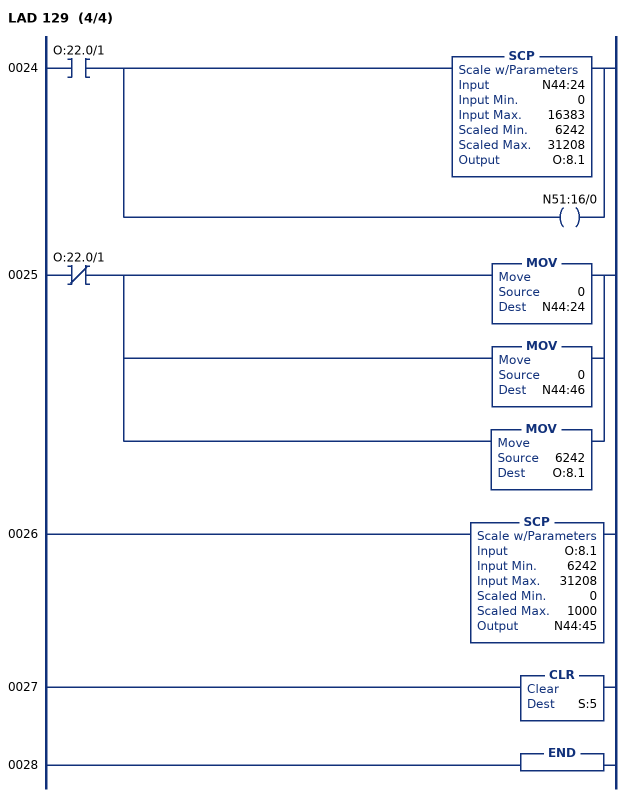
% Rung: 24 %
SOR XIC O:22.0/1 BST SCP N44:24 0 16383 6242 31208 O:8.1 NXB OTE N51:16/0 BND EOR
% Rung: 25 %
SOR XIO O:22.0/1 BST MOV 0 N44:24 NXB MOV 0 N44:46 NXB MOV 6242 O:8.1 BND EOR
% Rung: 26 %
SOR SCP O:8.1 6242 31208 0 1000 N44:45 EOR
% Rung: 27 %
SOR CLR S:5 EOR
% Rung: 28 %
SOR END EOR

LADDER 131
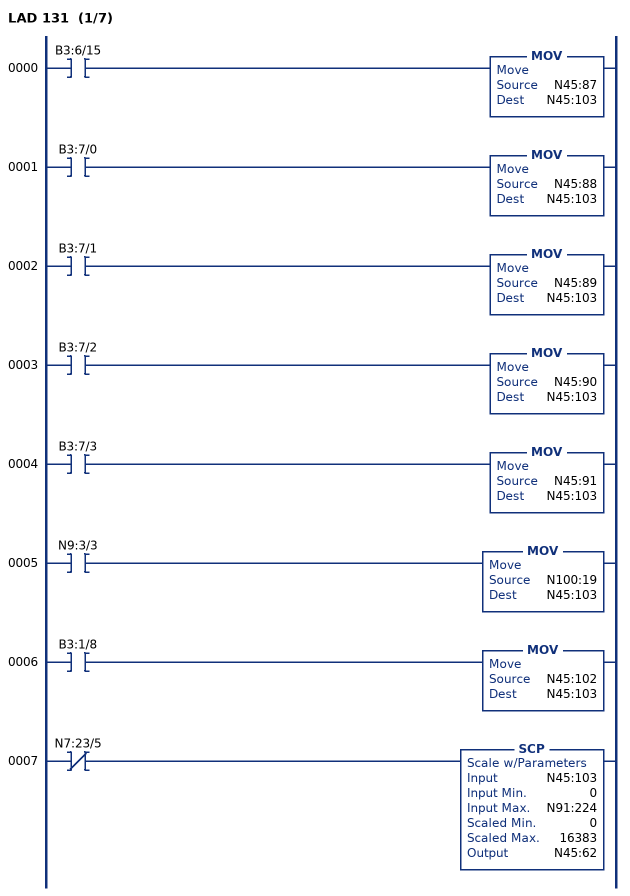
% Rung: 0 %
SOR XIC B3:6/15 MOV N45:87 N45:103 EOR
% Rung: 1 %
SOR XIC B3:7/0 MOV N45:88 N45:103 EOR
% Rung: 2 %
SOR XIC B3:7/1 MOV N45:89 N45:103 EOR
% Rung: 3 %
SOR XIC B3:7/2 MOV N45:90 N45:103 EOR
% Rung: 4 %
SOR XIC B3:7/3 MOV N45:91 N45:103 EOR
% Rung: 5 %
SOR XIC N9:3/3 MOV N100:19 N45:103 EOR
% Rung: 6 %
SOR XIC B3:1/8 MOV N45:102 N45:103 EOR
% Rung: 7 %
SOR XIO N7:23/5 SCP N45:103 0 N91:224 0 16383 N45:62 EOR

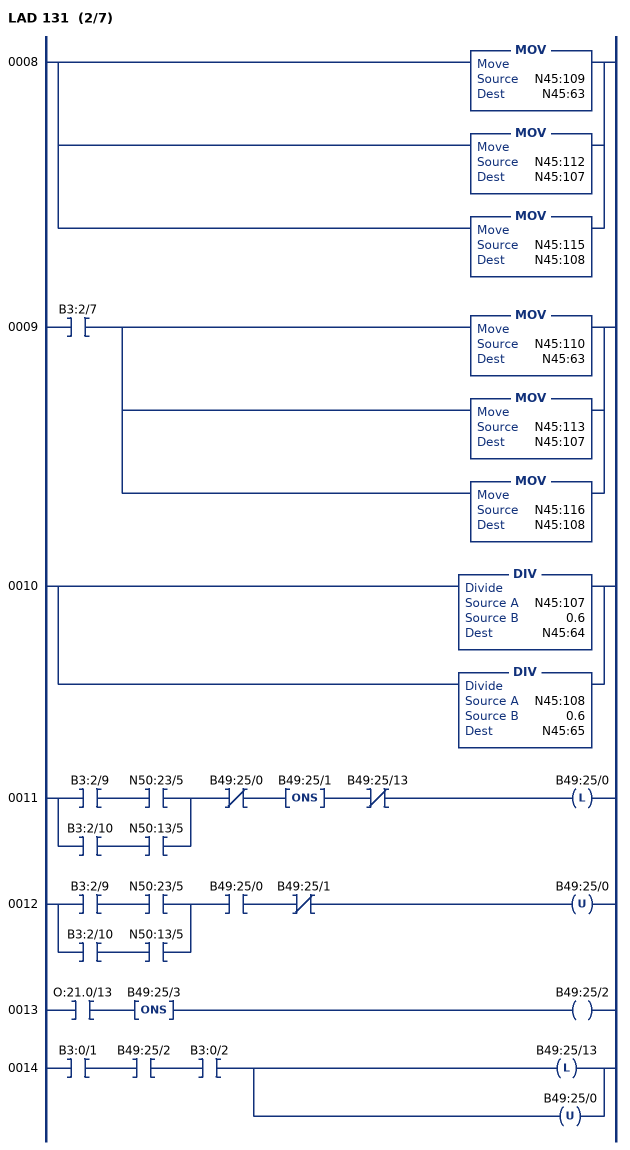
% Rung: 8 %
SOR BST MOV N45:109 N45:63 NXB MOV N45:112 N45:107 NXB MOV N45:115 N45:108 BND EOR
% Rung: 9 %
SOR XIC B3:2/7 BST MOV N45:110 N45:63 NXB MOV N45:113 N45:107 NXB MOV N45:116 N45:108 BND EOR
% Rung: 10 %
SOR BST DIV N45:107 0.6 N45:64 NXB DIV N45:108 0.6 N45:65 BND EOR
% Rung: 11 %
SOR BST XIC B3:2/9 XIC N50:23/5 NXB XIC B3:2/10 XIC N50:13/5 BND XIO B49:25/0 OSR B49:25/1 XIO B49:25/13 OTL B49:25/0 EOR
% Rung: 12 %
SOR BST XIC B3:2/9 XIC N50:23/5 NXB XIC B3:2/10 XIC N50:13/5 BND XIC B49:25/0 XIO B49:25/1 OTU B49:25/0 EOR
% Rung: 13 %
SOR XIC O:21.0/13 OSR B49:25/3 OTE B49:25/2 EOR
% Rung: 14 %
SOR XIC B3:0/1 XIC B49:25/2 XIC B3:0/2 BST OTL B49:25/13 NXB OTU B49:25/0 BND EOR

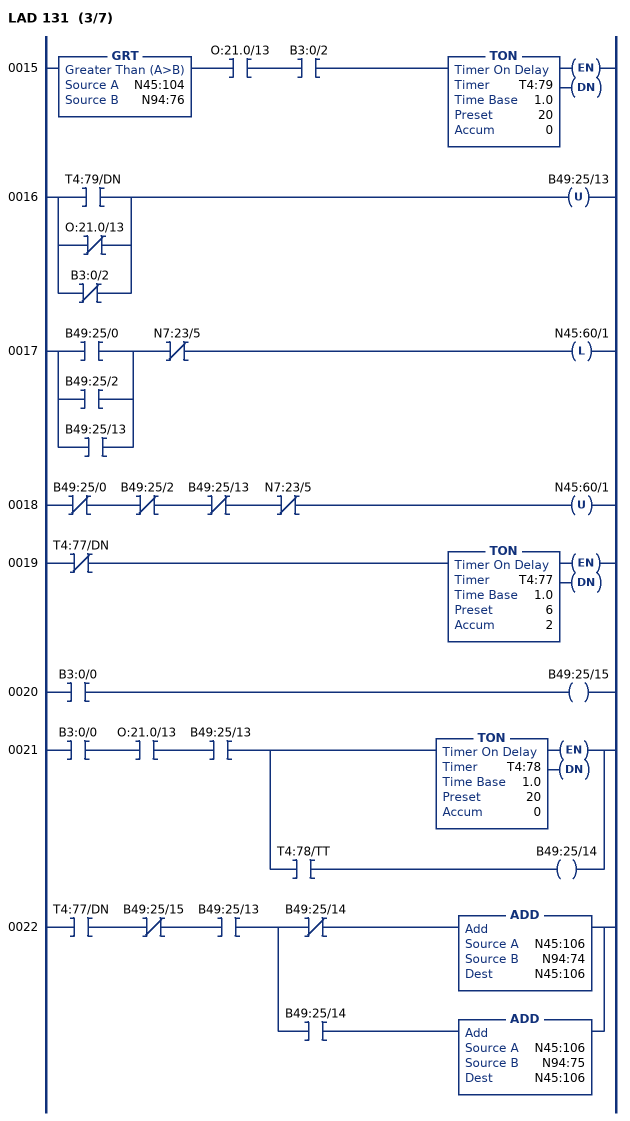
% Rung: 15 %
SOR GRT N45:104 N94:76 XIC O:21.0/13 XIC B3:0/2 TON T4:79 1.0 20 0 EOR
% Rung: 16 %
SOR BST XIC T4:79/DN NXB XIO O:21.0/13 NXB XIO B3:0/2 BND OTU B49:25/13 EOR
% Rung: 17 %
SOR BST XIC B49:25/0 NXB XIC B49:25/2 NXB XIC B49:25/13 BND XIO N7:23/5 OTL N45:60/1 EOR
% Rung: 18 %
SOR XIO B49:25/0 XIO B49:25/2 XIO B49:25/13 XIO N7:23/5 OTU N45:60/1 EOR
% Rung: 19 %
SOR XIO T4:77/DN TON T4:77 1.0 6 2 EOR
% Rung: 20 %
SOR XIC B3:0/0 OTE B49:25/15 EOR
% Rung: 21 %
SOR XIC B3:0/0 XIC O:21.0/13 XIC B49:25/13 BST TON T4:78 1.0 20 0 NXB XIC T4:78/TT OTE B49:25/14 BND EOR
% Rung: 22 %
SOR XIC T4:77/DN XIO B49:25/15 XIC B49:25/13 BST XIO B49:25/14 ADD N45:106 N94:74 N45:106 NXB XIC B49:25/14 ADD N45:106 N94:75 N45:106 BND EOR

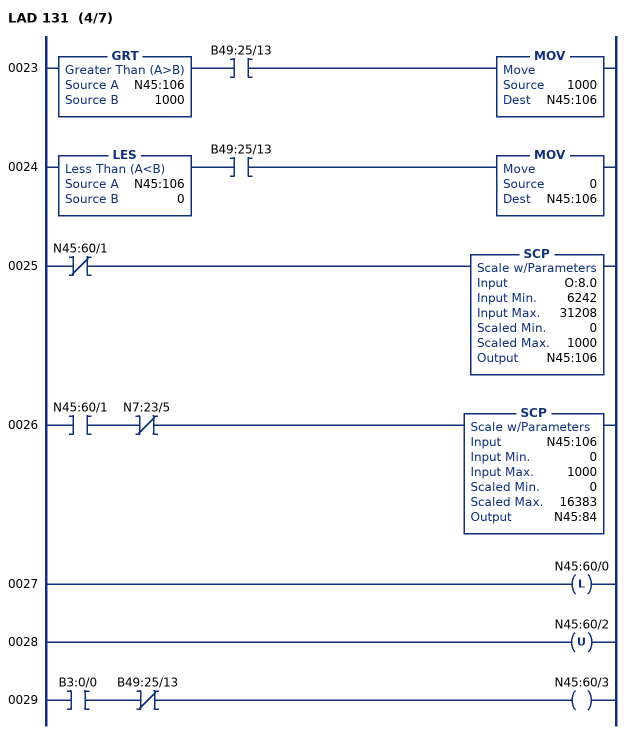
% Rung: 23 %
SOR GRT N45:106 1000 XIC B49:25/13 MOV 1000 N45:106 EOR
% Rung: 24 %
SOR LES N45:106 0 XIC B49:25/13 MOV 0 N45:106 EOR
% Rung: 25 %
SOR XIO N45:60/1 SCP O:8.0 6242 31208 0 1000 N45:106 EOR
% Rung: 26 %
SOR XIC N45:60/1 XIO N7:23/5 SCP N45:106 0 1000 0 16383 N45:84 EOR
% Rung: 27 %
SOR OTL N45:60/0 EOR
% Rung: 28 %
SOR OTU N45:60/2 EOR
% Rung: 29 %
SOR XIC B3:0/0 XIO B49:25/13 OTE N45:60/3 EOR

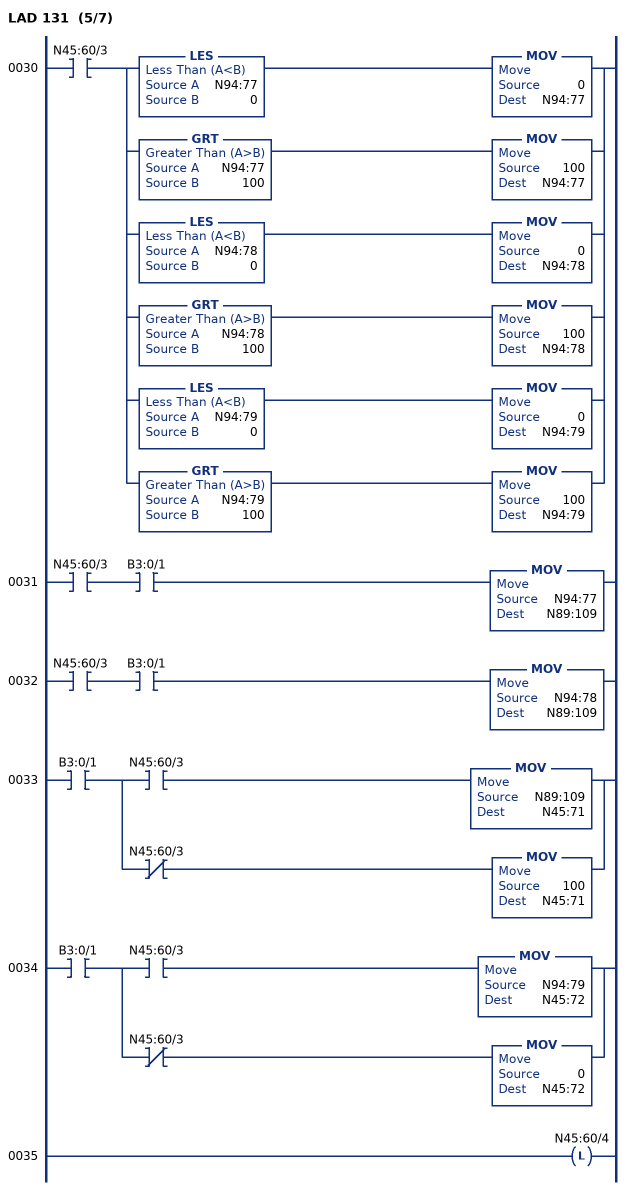
% Rung: 30 %
SOR XIC N45:60/3 BST LES N94:77 0 MOV 0 N94:77 NXB GRT N94:77 100 MOV 100 N94:77 NXB LES N94:78 0 MOV 0 N94:78 NXB GRT N94:78 100 MOV 100 N94:78 NXB LES N94:79 0 MOV 0 N94:79 NXB GRT N94:79 100 MOV 100 N94:79 BND EOR
% Rung: 31 %
SOR XIC N45:60/3 XIC B3:0/1 MOV N94:77 N89:109 EOR
% Rung: 32 %
SOR XIC N45:60/3 XIC B3:0/1 MOV N94:78 N89:109 EOR
% Rung: 33 %
SOR XIC B3:0/1 BST XIC N45:60/3 MOV N89:109 N45:71 NXB XIO N45:60/3 MOV 100 N45:71 BND EOR
% Rung: 34 %
SOR XIC B3:0/1 BST XIC N45:60/3 MOV N94:79 N45:72 NXB XIO N45:60/3 MOV 0 N45:72 BND EOR
% Rung: 35 %
SOR OTL N45:60/4 EOR

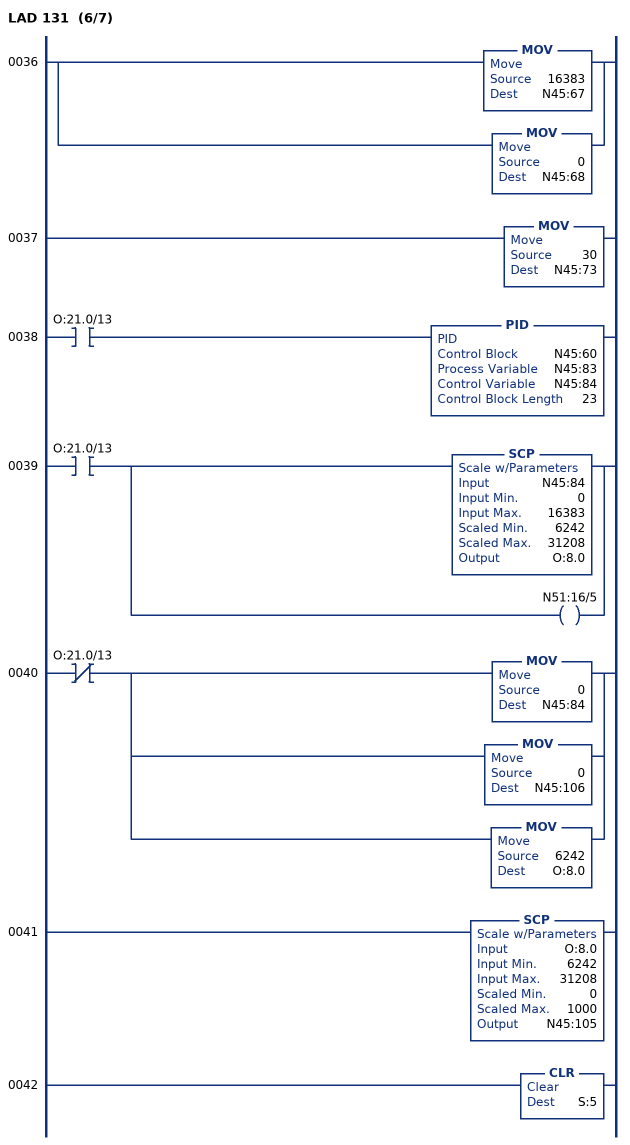
% Rung: 36 %
SOR BST MOV 16383 N45:67 NXB MOV 0 N45:68 BND EOR
% Rung: 37 %
SOR MOV 30 N45:73 EOR
% Rung: 38 %
SOR XIC O:21.0/13 PID N45:60 N45:83 N45:84 23 EOR
% Rung: 39 %
SOR XIC O:21.0/13 BST SCP N45:84 0 16383 6242 31208 O:8.0 NXB OTE N51:16/5 BND EOR
% Rung: 40 %
SOR XIO O:21.0/13 BST MOV 0 N45:84 NXB MOV 0 N45:106 NXB MOV 6242 O:8.0 BND EOR
% Rung: 41 %
SOR SCP O:8.0 6242 31208 0 1000 N45:105 EOR
% Rung: 42 %
SOR CLR S:5 EOR

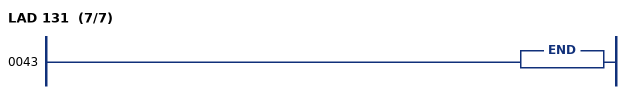
% Rung: 43 %
SOR END EOR

LADDER 132
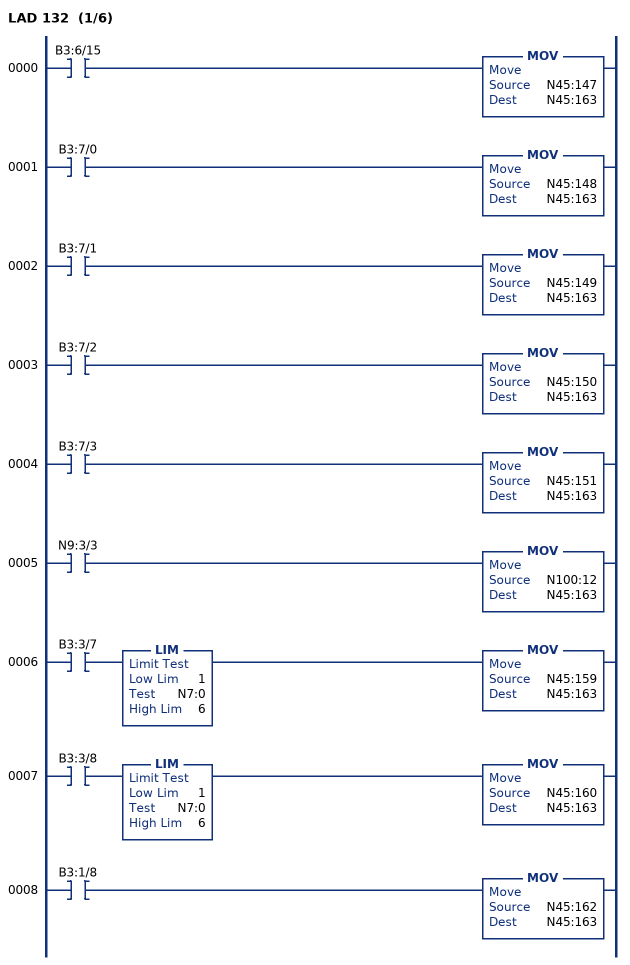
% Rung: 0 %
SOR XIC B3:6/15 MOV N45:147 N45:163 EOR
% Rung: 1 %
SOR XIC B3:7/0 MOV N45:148 N45:163 EOR
% Rung: 2 %
SOR XIC B3:7/1 MOV N45:149 N45:163 EOR
% Rung: 3 %
SOR XIC B3:7/2 MOV N45:150 N45:163 EOR
% Rung: 4 %
SOR XIC B3:7/3 MOV N45:151 N45:163 EOR
% Rung: 5 %
SOR XIC N9:3/3 MOV N100:12 N45:163 EOR
% Rung: 6 %
SOR XIC B3:3/7 LIM 1 N7:0 6 MOV N45:159 N45:163 EOR
% Rung: 7 %
SOR XIC B3:3/8 LIM 1 N7:0 6 MOV N45:160 N45:163 EOR
% Rung: 8 %
SOR XIC B3:1/8 MOV N45:162 N45:163 EOR

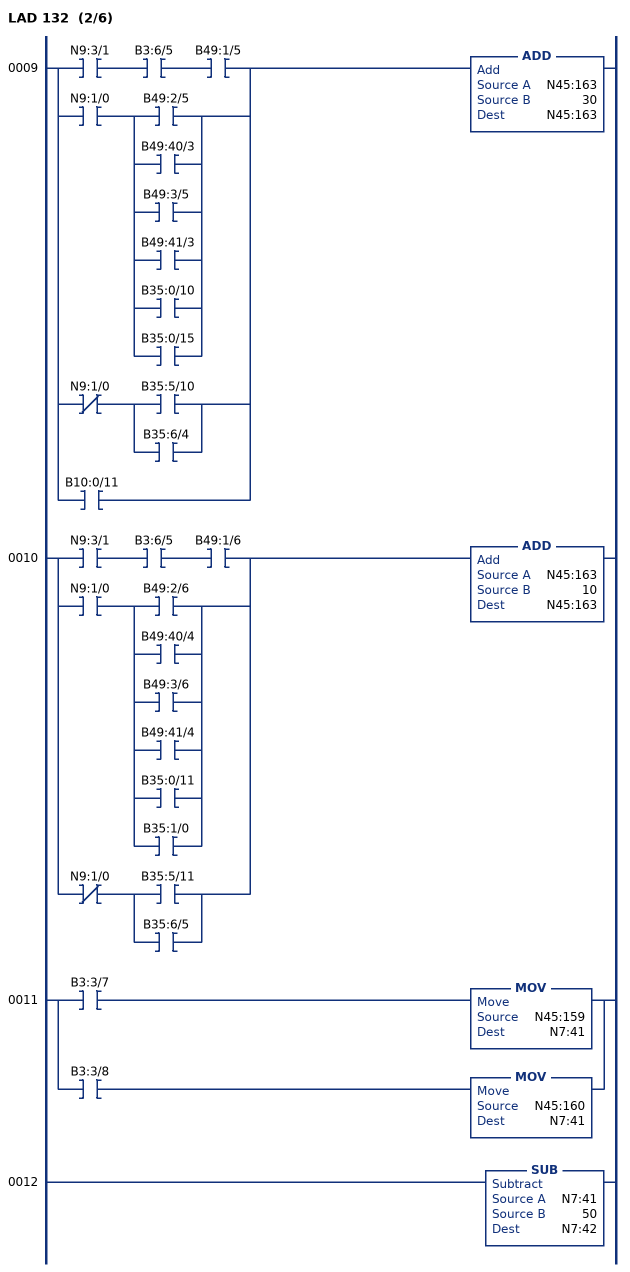
% Rung: 9 %
SOR BST XIC N9:3/1 XIC B3:6/5 XIC B49:1/5 NXB XIC N9:1/0 BST XIC B49:2/5 NXB XIC B49:40/3 NXB XIC B49:3/5 NXB XIC B49:41/3 NXB XIC B35:0/10 NXB XIC B35:0/15 BND NXB XIO N9:1/0 BST XIC B35:5/10 NXB XIC B35:6/4 BND NXB XIC B10:0/11 BND ADD N45:163 30 N45:163 EOR
% Rung: 10 %
SOR BST XIC N9:3/1 XIC B3:6/5 XIC B49:1/6 NXB XIC N9:1/0 BST XIC B49:2/6 NXB XIC B49:40/4 NXB XIC B49:3/6 NXB XIC B49:41/4 NXB XIC B35:0/11 NXB XIC B35:1/0 BND NXB XIO N9:1/0 BST XIC B35:5/11 NXB XIC B35:6/5 BND BND ADD N45:163 10 N45:163 EOR
% Rung: 11 %
SOR BST XIC B3:3/7 MOV N45:159 N7:41 NXB XIC B3:3/8 MOV N45:160 N7:41 BND EOR
% Rung: 12 %
SOR SUB N7:41 50 N7:42 EOR

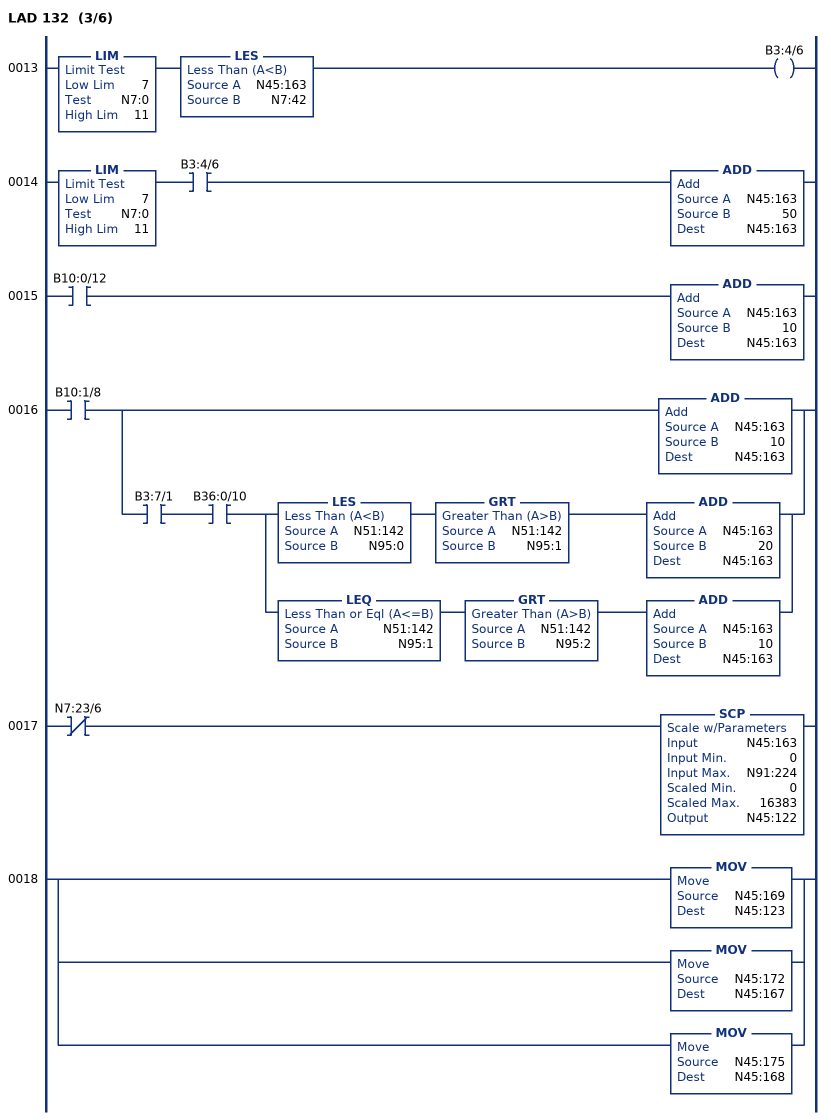
% Rung: 13 %
SOR LIM 7 N7:0 11 LES N45:163 N7:42 OTE B3:4/6 EOR
% Rung: 14 %
SOR LIM 7 N7:0 11 XIC B3:4/6 ADD N45:163 50 N45:163 EOR
% Rung: 15 %
SOR XIC B10:0/12 ADD N45:163 10 N45:163 EOR
% Rung: 16 %
SOR XIC B10:1/8 BST ADD N45:163 10 N45:163 NXB XIC B3:7/1 XIC B36:0/10 BST LES N51:142 N95:0 GRT N51:142 N95:1 ADD N45:163 20 N45:163 NXB LEQ N51:142 N95:1 GRT N51:142 N95:2 ADD N45:163 10 N45:163 BND BND EOR
% Rung: 17 %
SOR XIO N7:23/6 SCP N45:163 0 N91:224 0 16383 N45:122 EOR
% Rung: 18 %
SOR BST MOV N45:169 N45:123 NXB MOV N45:172 N45:167 NXB MOV N45:175 N45:168 BND EOR

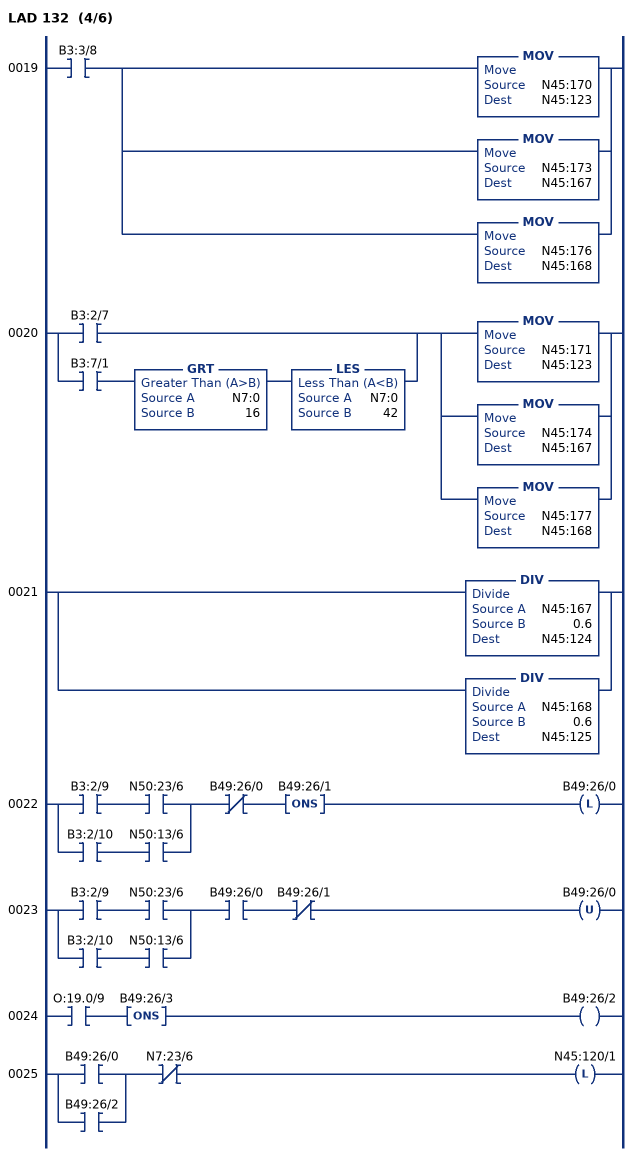
% Rung: 19 %
SOR XIC B3:3/8 BST MOV N45:170 N45:123 NXB MOV N45:173 N45:167 NXB MOV N45:176 N45:168 BND EOR
% Rung: 20 %
SOR BST XIC B3:2/7 NXB XIC B3:7/1 GRT N7:0 16 LES N7:0 42 BND BST MOV N45:171 N45:123 NXB MOV N45:174 N45:167 NXB MOV N45:177 N45:168 BND EOR
% Rung: 21 %
SOR BST DIV N45:167 0.6 N45:124 NXB DIV N45:168 0.6 N45:125 BND EOR
% Rung: 22 %
SOR BST XIC B3:2/9 XIC N50:23/6 NXB XIC B3:2/10 XIC N50:13/6 BND XIO B49:26/0 OSR B49:26/1 OTL B49:26/0 EOR
% Rung: 23 %
SOR BST XIC B3:2/9 XIC N50:23/6 NXB XIC B3:2/10 XIC N50:13/6 BND XIC B49:26/0 XIO B49:26/1 OTU B49:26/0 EOR
% Rung: 24 %
SOR XIC O:19.0/9 OSR B49:26/3 OTE B49:26/2 EOR
% Rung: 25 %
SOR BST XIC B49:26/0 NXB XIC B49:26/2 BND XIO N7:23/6 OTL N45:120/1 EOR

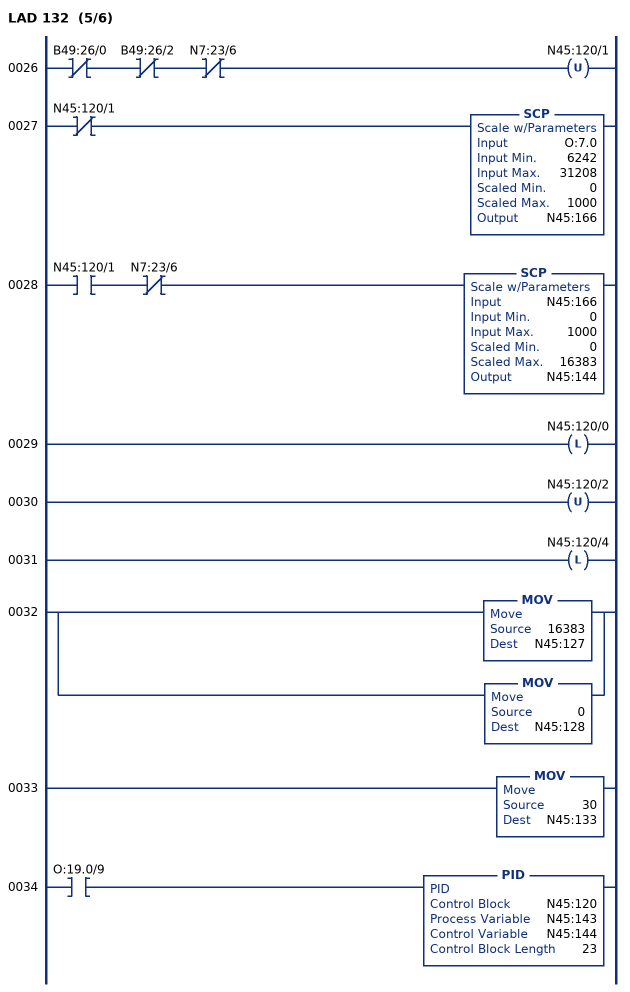
% Rung: 26 %
SOR XIO B49:26/0 XIO B49:26/2 XIO N7:23/6 OTU N45:120/1 EOR
% Rung: 27 %
SOR XIO N45:120/1 SCP O:7.0 6242 31208 0 1000 N45:166 EOR
% Rung: 28 %
SOR XIC N45:120/1 XIO N7:23/6 SCP N45:166 0 1000 0 16383 N45:144 EOR
% Rung: 29 %
SOR OTL N45:120/0 EOR
% Rung: 30 %
SOR OTU N45:120/2 EOR
% Rung: 31 %
SOR OTL N45:120/4 EOR
% Rung: 32 %
SOR BST MOV 16383 N45:127 NXB MOV 0 N45:128 BND EOR
% Rung: 33 %
SOR MOV 30 N45:133 EOR
% Rung: 34 %
SOR XIC O:19.0/9 PID N45:120 N45:143 N45:144 23 EOR

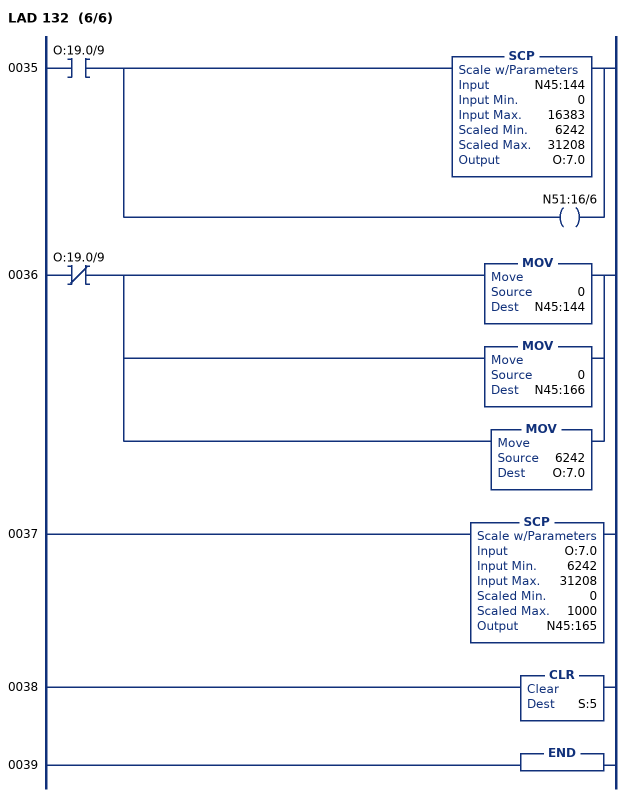
% Rung: 35 %
SOR XIC O:19.0/9 BST SCP N45:144 0 16383 6242 31208 O:7.0 NXB OTE N51:16/6 BND EOR
% Rung: 36 %
SOR XIO O:19.0/9 BST MOV 0 N45:144 NXB MOV 0 N45:166 NXB MOV 6242 O:7.0 BND EOR
% Rung: 37 %
SOR SCP O:7.0 6242 31208 0 1000 N45:165 EOR
% Rung: 38 %
SOR CLR S:5 EOR
% Rung: 39 %
SOR END EOR

LADDER 133
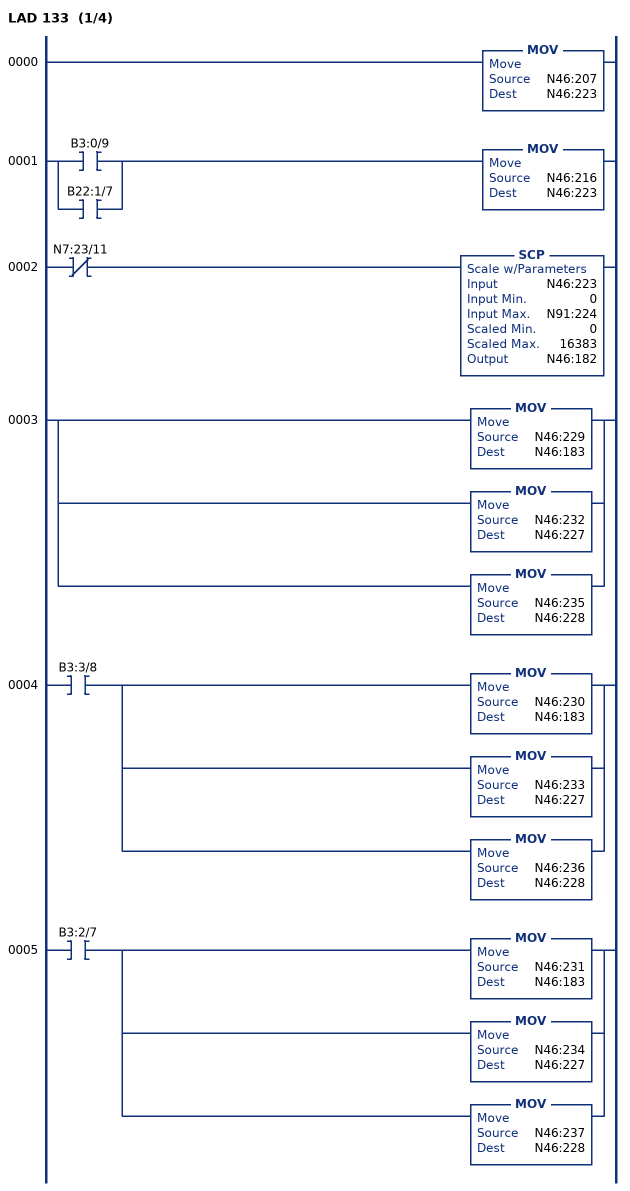
% Rung: 0 %
SOR MOV N46:207 N46:223 EOR
% Rung: 1 %
SOR BST XIC B3:0/9 NXB XIC B22:1/7 BND MOV N46:216 N46:223 EOR
% Rung: 2 %
SOR XIO N7:23/11 SCP N46:223 0 N91:224 0 16383 N46:182 EOR
% Rung: 3 %
SOR BST MOV N46:229 N46:183 NXB MOV N46:232 N46:227 NXB MOV N46:235 N46:228 BND EOR
% Rung: 4 %
SOR XIC B3:3/8 BST MOV N46:230 N46:183 NXB MOV N46:233 N46:227 NXB MOV N46:236 N46:228 BND EOR
% Rung: 5 %
SOR XIC B3:2/7 BST MOV N46:231 N46:183 NXB MOV N46:234 N46:227 NXB MOV N46:237 N46:228 BND EOR

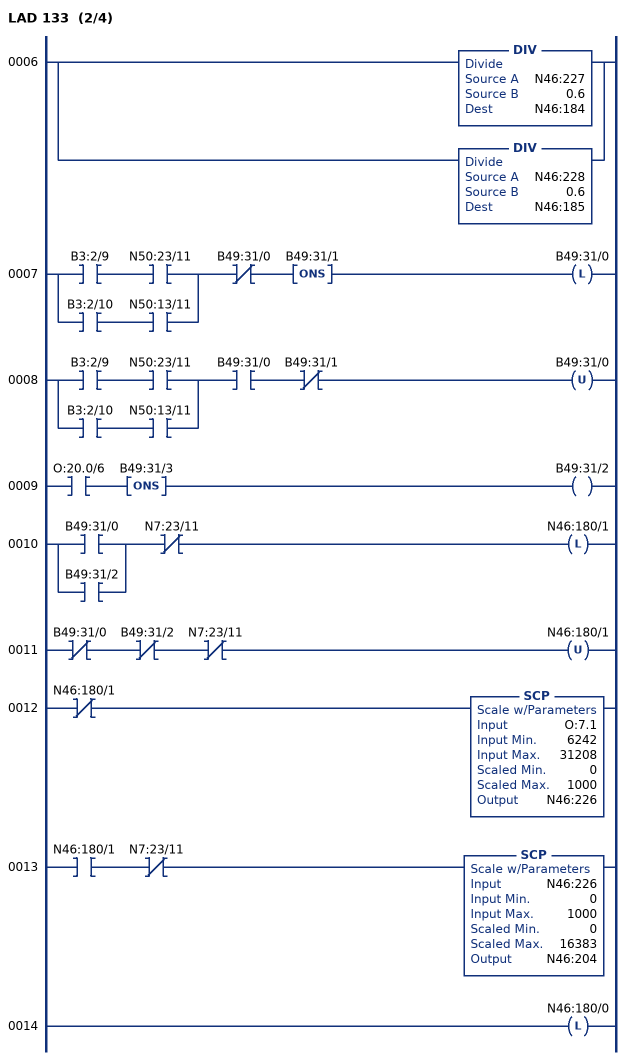
% Rung: 6 %
SOR BST DIV N46:227 0.6 N46:184 NXB DIV N46:228 0.6 N46:185 BND EOR
% Rung: 7 %
SOR BST XIC B3:2/9 XIC N50:23/11 NXB XIC B3:2/10 XIC N50:13/11 BND XIO B49:31/0 OSR B49:31/1 OTL B49:31/0 EOR
% Rung: 8 %
SOR BST XIC B3:2/9 XIC N50:23/11 NXB XIC B3:2/10 XIC N50:13/11 BND XIC B49:31/0 XIO B49:31/1 OTU B49:31/0 EOR
% Rung: 9 %
SOR XIC O:20.0/6 OSR B49:31/3 OTE B49:31/2 EOR
% Rung: 10 %
SOR BST XIC B49:31/0 NXB XIC B49:31/2 BND XIO N7:23/11 OTL N46:180/1 EOR
% Rung: 11 %
SOR XIO B49:31/0 XIO B49:31/2 XIO N7:23/11 OTU N46:180/1 EOR
% Rung: 12 %
SOR XIO N46:180/1 SCP O:7.1 6242 31208 0 1000 N46:226 EOR
% Rung: 13 %
SOR XIC N46:180/1 XIO N7:23/11 SCP N46:226 0 1000 0 16383 N46:204 EOR
% Rung: 14 %
SOR OTL N46:180/0 EOR

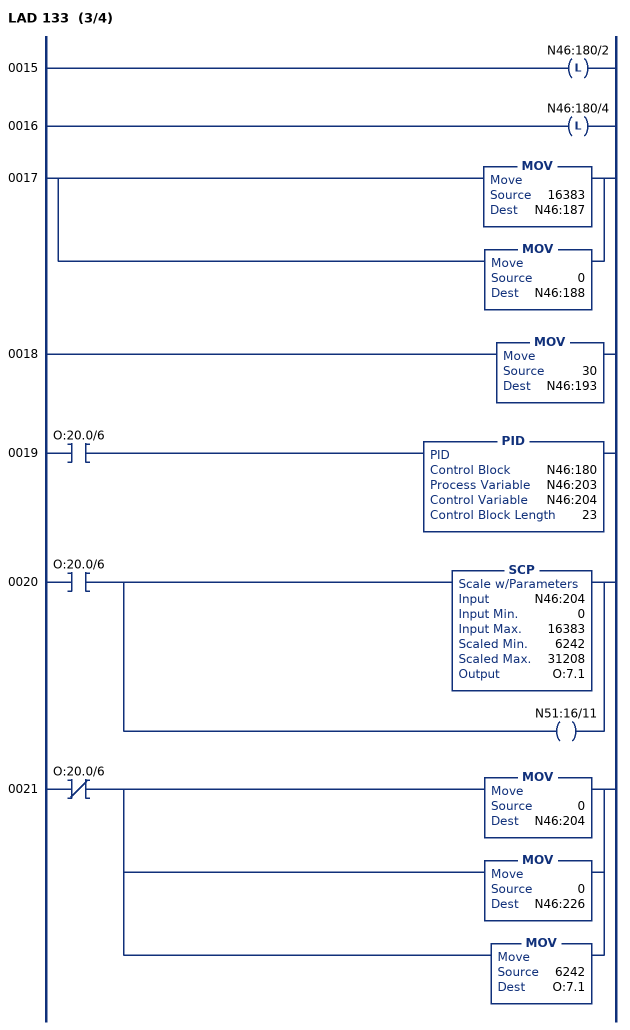
% Rung: 15 %
SOR OTL N46:180/2 EOR
% Rung: 16 %
SOR OTL N46:180/4 EOR
% Rung: 17 %
SOR BST MOV 16383 N46:187 NXB MOV 0 N46:188 BND EOR
% Rung: 18 %
SOR MOV 30 N46:193 EOR
% Rung: 19 %
SOR XIC O:20.0/6 PID N46:180 N46:203 N46:204 23 EOR
% Rung: 20 %
SOR XIC O:20.0/6 BST SCP N46:204 0 16383 6242 31208 O:7.1 NXB OTE N51:16/11 BND EOR
% Rung: 21 %
SOR XIO O:20.0/6 BST MOV 0 N46:204 NXB MOV 0 N46:226 NXB MOV 6242 O:7.1 BND EOR

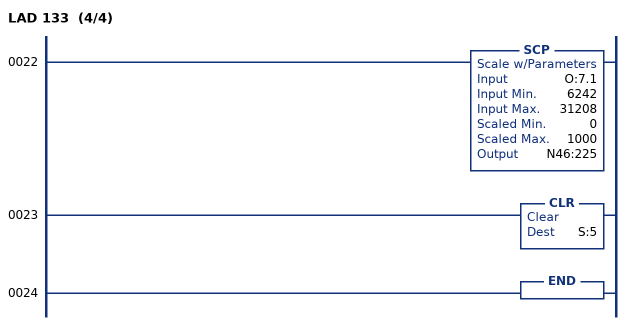
% Rung: 22 %
SOR SCP O:7.1 6242 31208 0 1000 N46:225 EOR
% Rung: 23 %
SOR CLR S:5 EOR
% Rung: 24 %
SOR END EOR

LADDER 134
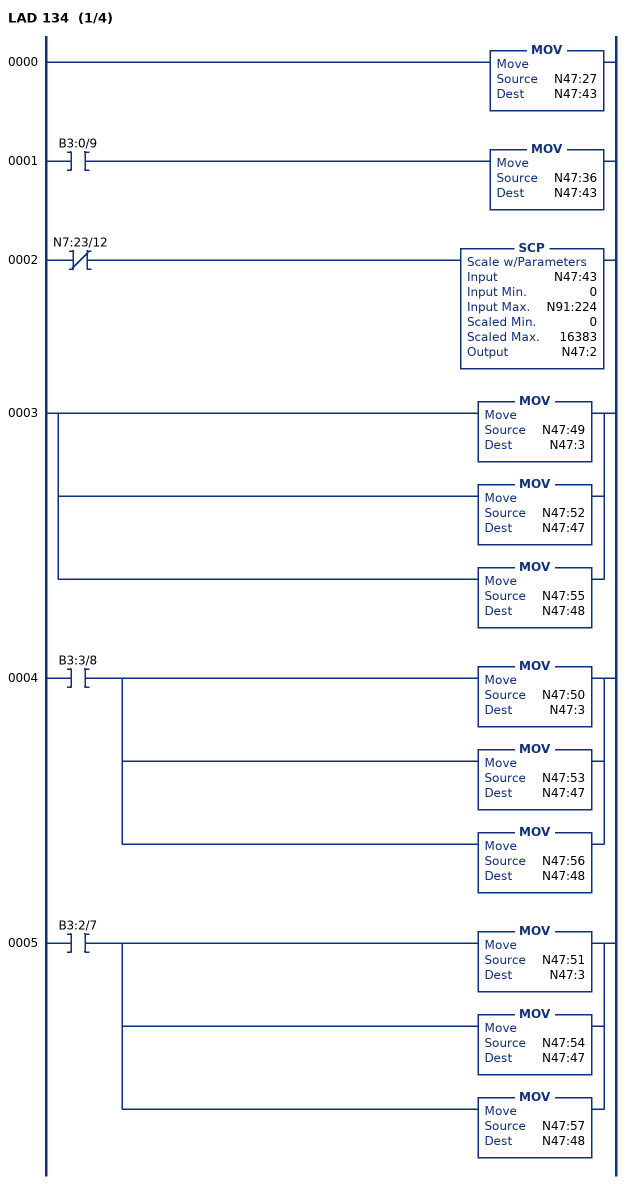
% Rung: 0 %
SOR MOV N47:27 N47:43 EOR
% Rung: 1 %
SOR XIC B3:0/9 MOV N47:36 N47:43 EOR
% Rung: 2 %
SOR XIO N7:23/12 SCP N47:43 0 N91:224 0 16383 N47:2 EOR
% Rung: 3 %
SOR BST MOV N47:49 N47:3 NXB MOV N47:52 N47:47 NXB MOV N47:55 N47:48 BND EOR
% Rung: 4 %
SOR XIC B3:3/8 BST MOV N47:50 N47:3 NXB MOV N47:53 N47:47 NXB MOV N47:56 N47:48 BND EOR
% Rung: 5 %
SOR XIC B3:2/7 BST MOV N47:51 N47:3 NXB MOV N47:54 N47:47 NXB MOV N47:57 N47:48 BND EOR

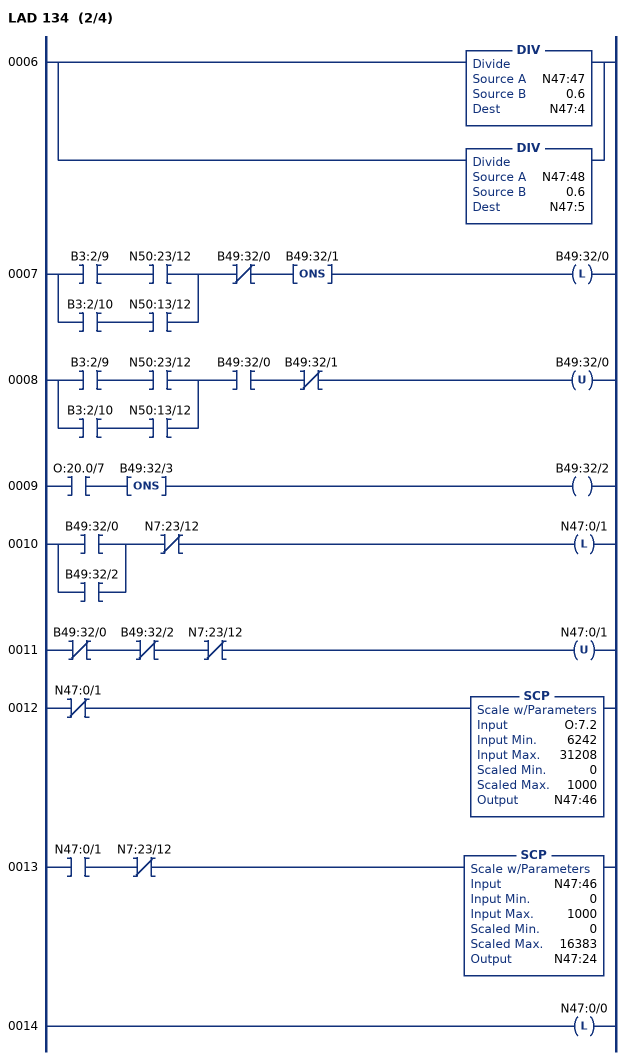
% Rung: 6 %
SOR BST DIV N47:47 0.6 N47:4 NXB DIV N47:48 0.6 N47:5 BND EOR
% Rung: 7 %
SOR BST XIC B3:2/9 XIC N50:23/12 NXB XIC B3:2/10 XIC N50:13/12 BND XIO B49:32/0 OSR B49:32/1 OTL B49:32/0 EOR
% Rung: 8 %
SOR BST XIC B3:2/9 XIC N50:23/12 NXB XIC B3:2/10 XIC N50:13/12 BND XIC B49:32/0 XIO B49:32/1 OTU B49:32/0 EOR
% Rung: 9 %
SOR XIC O:20.0/7 OSR B49:32/3 OTE B49:32/2 EOR
% Rung: 10 %
SOR BST XIC B49:32/0 NXB XIC B49:32/2 BND XIO N7:23/12 OTL N47:0/1 EOR
% Rung: 11 %
SOR XIO B49:32/0 XIO B49:32/2 XIO N7:23/12 OTU N47:0/1 EOR
% Rung: 12 %
SOR XIO N47:0/1 SCP O:7.2 6242 31208 0 1000 N47:46 EOR
% Rung: 13 %
SOR XIC N47:0/1 XIO N7:23/12 SCP N47:46 0 1000 0 16383 N47:24 EOR
% Rung: 14 %
SOR OTL N47:0/0 EOR

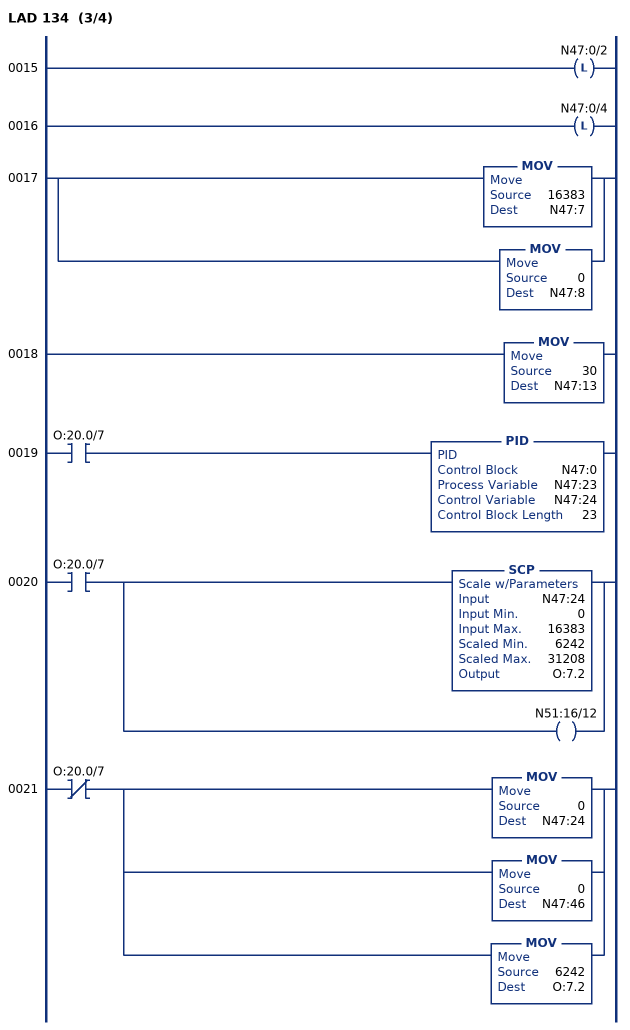
% Rung: 15 %
SOR OTL N47:0/2 EOR
% Rung: 16 %
SOR OTL N47:0/4 EOR
% Rung: 17 %
SOR BST MOV 16383 N47:7 NXB MOV 0 N47:8 BND EOR
% Rung: 18 %
SOR MOV 30 N47:13 EOR
% Rung: 19 %
SOR XIC O:20.0/7 PID N47:0 N47:23 N47:24 23 EOR
% Rung: 20 %
SOR XIC O:20.0/7 BST SCP N47:24 0 16383 6242 31208 O:7.2 NXB OTE N51:16/12 BND EOR
% Rung: 21 %
SOR XIO O:20.0/7 BST MOV 0 N47:24 NXB MOV 0 N47:46 NXB MOV 6242 O:7.2 BND EOR

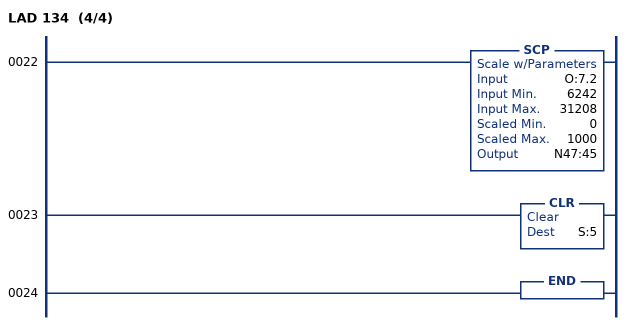
% Rung: 22 %
SOR SCP O:7.2 6242 31208 0 1000 N47:45 EOR
% Rung: 23 %
SOR CLR S:5 EOR
% Rung: 24 %
SOR END EOR

DATA TABLE (non-zero values as saved)
DATA B3
% B3:0 % 0X0002 0X0841 0X0300 0X0084 0X3F80 0X8000 0X8540 0X0000 0X0000 0X0000
% B3:10 % 0X0001 0X0000 0X0000 0X0000 0X0000 0X0000 0X0000 0X0000 0X0000 0X0401
% B3:20 % 0X0000 0X0000 0X0000 0X0000 0X0000 0X00A6 0X0000 0X0000 0X0000 0X0000
% B3:40 % 0X0000 0X0001 0X0000 0X0000 0X0000 0X0000 0X0000 0X0000 0X0000 0X0000
% B3:60 % 0X0000 0X0004 0X0020 0X0000 0X0800 0X0002 0X0000 0X00FE 0X0000 0X0000
% B3:70 % 0X0040 0X0000 0X8000 0X0001 0X0000 0X0000 0X0000 0X0000 0X0000 0X0000
% B3:120 % 0X0000 0X0000 0X0000 0X0000 0X0000 0X0000 0X8000 0X0000 0X0000 0X0000
DATA T4
% .PRE .ACC %
% T4:1 % 15 13
% T4:3 % 50 38
% T4:4 % 50 0
% T4:5 % 15 0
% T4:6 % 60 0
% T4:7 % 120 120
% T4:8 % 3600 0
% T4:9 % 30000 0
% T4:10 % 30 0
% T4:11 % 500 0
% T4:12 % 10 0
% T4:13 % 10 0
% T4:14 % 200 0
% T4:15 % 60 0
% T4:16 % 50 0
% T4:17 % 100 0
% T4:18 % 30 0
% T4:20 % 1 0
% T4:21 % 60 20
% T4:22 % 3 3
% T4:25 % 25 0
% T4:26 % 30 0
% T4:30 % 25 25
% T4:31 % 10 0
% T4:32 % 5 5
% T4:33 % 300 0
% T4:34 % 30 0
% T4:35 % 1 0
% T4:36 % 30 0
% T4:37 % 10 0
% T4:38 % 1 0
% T4:40 % 20 0
% T4:41 % 20 0
% T4:42 % 200 0
% T4:43 % 100 100
% T4:44 % 50 0
% T4:49 % 30 0
% T4:50 % 1 0
% T4:51 % 20 0
% T4:52 % 6 5
% T4:53 % 20 0
% T4:54 % 20 20
% T4:55 % 1 0
% T4:56 % 20 0
% T4:60 % 150 0
% T4:61 % 20 0
% T4:65 % 1 0
% T4:66 % 20 0
% T4:72 % 6 6
% T4:73 % 20 0
% T4:74 % 20 0
% T4:75 % 20 0
% T4:77 % 6 2
% T4:78 % 20 0
% T4:79 % 20 0
% T4:80 % 1 0
% T4:81 % 20 0
% T4:85 % 1 0
% T4:86 % 20 0
% T4:90 % 1 0
% T4:91 % 20 0
% T4:92 % 1 0
% T4:93 % 20 0
% T4:100 % 1 0
% T4:101 % 20 0
% T4:111 % 120 0
% T4:112 % 6 6
% T4:113 % 20 0
% T4:114 % 20 0
% T4:115 % 222 0
% T4:116 % 6 6
% T4:117 % 20 0
% T4:119 % 60 0
% T4:120 % 6 6
% T4:121 % 20 0
DATA C5
% .PRE .ACC %
% C5:0 % 4 0
% C5:1 % 2 0
% C5:4 % 2 0
% C5:5 % 3 0
DATA R6
% .LEN .POS %
% R6:0 % 3 0
% R6:1 % 4 0
% R6:2 % 4 0
% R6:3 % 3 0
% R6:4 % 14 0
% R6:5 % 14 0
% R6:6 % 14 0
% R6:7 % 14 0
% R6:8 % 14 0
% R6:9 % 14 0
% R6:10 % 14 0
% R6:11 % 14 0
DATA N7
% N7:0 % 0 514 200 0 0 11 101 10 0 0
% N7:10 % 0 514 200 0 0 0 0 0 0 0
% N7:30 % 1390 0 0 0 0 0 0 0 0 0
% N7:40 % -1 1380 1330 0 0 0 0 0 0 0
% N7:50 % 0 14 0
DATA F8
% F8:0 % 237.777 0 0 0 0
% F8:5 % 0 0.01 0 0 0
% F8:10 % 1 770 1 900 1
% F8:15 % 950 0 0 1 1000
% F8:20 % 1 820 1 0 0.7076923
% F8:25 % 0 1.25 630 0.7076923 0
% F8:30 % 1 1000 1 0 1
% F8:35 % 0 1 0 2 150
% F8:40 % 17.87234 0 0 0 0
DATA N9
% N9:0 % 18434 2683 699 4243 0 0 0 0 0 2
% N9:10 % 2957 0 0 0
DATA B10
% B10:0 % 0X0001 0X0000 0X0000 0X0000 0X0000 0X0000 0X0000 0X0000 0X0000 0X0000
DATA B11
% B11:0 % 0X0001 0X0000 0X0000 0X0000 0X0000 0X0000 0X0000 0X0000 0X0000 0X0000
% B11:30 % 0X0000 0X0000 0X0004
DATA B12
% B12:0 % 0X0001 0X0000 0X0000 0X0000 0X0000 0X0000 0X0000 0X0000 0X0000 0X0000
% B12:10 % 0X0000 0X0000 0X0100 0X0000
DATA B18
% B18:0 % 0X0000 0X0010 0X0000 0X0000
DATA T21
% .PRE .ACC %
% T21:1 % 5 0
% T21:2 % 5 0
% T21:3 % 5 0
% T21:4 % 5 0
% T21:5 % 5 0
% T21:6 % 25 0
% T21:7 % 5 0
% T21:8 % 5 0
% T21:9 % 5 0
% T21:10 % 5 0
% T21:11 % 5 0
% T21:12 % 5 0
% T21:13 % 5 0
% T21:14 % 5 0
% T21:15 % 15 0
% T21:16 % 5 0
% T21:17 % 1000 0
% T21:18 % 600 0
% T21:19 % 10 0
% T21:20 % 10 0
% T21:21 % 300 0
% T21:22 % 1200 0
% T21:23 % 300 0
% T21:24 % 5 0
% T21:25 % 1 0
% T21:27 % 15 0
% T21:28 % 15 0
% T21:29 % 15 0
% T21:30 % 15 0
% T21:31 % 1200 0
% T21:32 % 600 0
% T21:33 % 300 0
% T21:34 % 15 0
% T21:35 % 1 0
% T21:36 % 10 0
% T21:37 % 600 0
% T21:38 % 180 0
% T21:40 % 600 0
% T21:41 % 20 0
% T21:42 % 10 0
% T21:43 % 120 0
% T21:44 % 120 0
% T21:45 % 60 0
% T21:46 % 1 1
% T21:47 % 5 0
% T21:48 % 1 1
% T21:49 % 1 1
% T21:50 % 120 0
% T21:51 % 10 0
% T21:52 % 10 0
% T21:53 % 5 0
% T21:54 % 50 54
% T21:55 % 50 50
% T21:56 % 50 50
% T21:57 % 50 50
% T21:58 % 50 50
% T21:59 % 50 50
% T21:61 % 10 0
% T21:62 % 2 0
% T21:63 % 4 0
% T21:70 % 2 0
% T21:71 % 5 0
% T21:72 % 5 0
% T21:73 % 5 0
% T21:74 % 600 0
% T21:75 % 20 0
% T21:76 % 5 0
% T21:77 % 5 0
% T21:78 % 5 0
% T21:79 % 5 0
% T21:80 % 5 0
% T21:81 % 15 0
% T21:84 % 5 0
DATA B24
% B24:0 % 0X0000 0X0000 0X0000 0X0004 0X0000 0X0000 0X0010 0X0000
DATA N25
% N25:0 % 244 1350 1350 1000 1350 1330 1330 1300 1100 0
% N25:20 % 294 1250 1250 1100 500 450 350 350 950 400
% N25:40 % 0 950 950 950 950 950 950 0 0 0
% N25:60 % 0 950 950 950 950 950 950 0 0 0
% N25:80 % 0 950 950 950 950 950 950 0 0 0
% N25:100 % 0 100 0 0 0 0 0 0 0 0
% N25:110 % 1 50 50 400 300 400 0 0 0 0
% N25:120 % 0 0 0 15400 14600 900 700 0 0 0
% N25:130 % 0 0 0 20426 20326 0 0 0 0 0
% N25:140 % 300 0 0 0 0 0 0 0 0 0
DATA T31
% .PRE .ACC %
% T31:0 % 200 0
% T31:1 % 200 0
% T31:2 % 200 0
% T31:3 % 200 0
% T31:4 % 100 0
% T31:5 % 200 0
% T31:6 % 200 0
% T31:7 % 5 0
% T31:8 % 1 0
% T31:9 % 1 0
% T31:10 % 25 0
% T31:11 % 60 0
% T31:12 % 20 0
% T31:13 % 300 0
% T31:14 % 5 0
% T31:15 % 20 0
% T31:16 % 60 0
% T31:17 % 180 0
% T31:18 % 60 0
% T31:19 % 5 5
% T31:20 % 15 0
% T31:21 % 30 30
% T31:22 % 5 5
% T31:23 % 5 5
% T31:24 % 1 0
% T31:25 % 10 10
% T31:26 % 200 0
% T31:27 % 10 0
% T31:28 % 900 0
% T31:29 % 100 0
% T31:30 % 30 0
% T31:31 % 10 0
% T31:32 % 10 0
% T31:33 % 30 0
% T31:34 % 20 0
% T31:35 % 200 0
% T31:36 % 15 0
% T31:37 % 60 0
% T31:38 % 10 0
% T31:39 % 20 0
% T31:40 % 5 0
% T31:41 % 10 0
% T31:42 % 5 0
% T31:43 % 30 0
DATA N32
% N32:0 % 0 0 0 3791 4000 4000 0 2080 0 0
% N32:10 % 0 0 0 5000 0 0 4000 5000 0 0
% N32:20 % 5899 7734 0 0 17000 0 0 0 0 0
% N32:30 % 0 0 0 6242 6242 6242 0 6242 6242 6242
% N32:40 % 0 6242 7490 6242 0 0 0 0 0 0
% N32:100 % 0 2957 2957 2957 2957 0 0 2957 2957 2957
% N32:110 % 2957 0 2957 0 2957 2957 2957 2957 0 0
% N32:120 % 0 0 2957 0 0 0 0 0 2957 2957
% N32:130 % 2957 2957 2957 2957 2957 2957 2957
DATA B36
% B36:0 % 0X0410 0X0000
DATA N40
% N40:0 % -32239 21248 14028 152 250 0 0 16383 0 0
% N40:10 % 0 30 5 30 2291 11737 100 -16 -68 0
% N40:20 % -28880 9190 14028 0 16383 0 0 13000 11000 10000
% N40:30 % 8000 7000 6500 0 0 0 0 0 13000 6500
% N40:40 % 0 14000 14000 1370 0 1000 1000 150 0 100
% N40:50 % 120 0 40 15 0 0 0 0 0 0
% N40:60 % 17 0 0 100 58 0 0 16383 0 0
% N40:70 % 0 30 5 30 0 0 0 0 0 0
% N40:80 % 0 0 0 0 0 0 0 15000 11000 10000
% N40:90 % 6600 7000 6500 0 8000 0 0 0 15000 8300
% N40:100 % 8000 20000 14000 0 0 0 0 35 0 100
% N40:110 % 120 100 35 35 40 0 0 0 0 0
% N40:120 % -31727 21248 1122 0 0 0 0 16383 0 0
% N40:130 % 0 30 5 30 3277 -2155 0 0 0 0
% N40:140 % -13104 10140 1122 0 0 0 0 13000 11000 10000
% N40:150 % 8000 7000 6500 0 0 0 0 200 6500 6500
% N40:160 % 0 14000 14000 15000 0 0 0 0 0 100
% N40:170 % 120 0 40 15 0 0 0 0 0 0
% N40:180 % 529 21248 1122 0 0 0 0 16383 0 0
% N40:190 % 0 30 5 30 2291 11737 100 0 0 0
% N40:200 % 0 9190 14028 0 0 0 0 13000 11000 10000
% N40:210 % 8000 7000 6500 0 0 0 0 200 6500 6500
% N40:220 % 0 14000 14000 13000 0 0 0 0 0 100
% N40:230 % 120 0 40 15 0 0 0 0 0 0
DATA N41
% N41:0 % -32239 21248 14028 152 250 0 0 16383 0 0
% N41:10 % 0 30 5 30 2291 11737 100 -16 -68 0
% N41:20 % -28880 9190 14028 2291 16383 0 0 14000 12000 11000
% N41:30 % 9000 8000 7500 0 0 0 0 0 7500 7500
% N41:40 % 0 15000 15000 1370 224 1000 1000 150 0 100
% N41:50 % 120 0 40 15 0 0 0 0 0 0
% N41:60 % -32239 21248 14028 152 250 0 0 16383 0 0
% N41:70 % 0 30 5 30 2291 11737 100 -16 -68 0
% N41:80 % -28880 9190 14028 2291 16383 0 0 14000 12000 11000
% N41:90 % 9000 8000 7500 0 0 0 15000 0 7500 7500
% N41:100 % 0 15000 15000 1370 224 1000 1000 150 0 100
% N41:110 % 120 0 40 15 0 0 0 0 0 0
% N41:120 % -32239 21248 14028 152 250 0 0 16383 0 0
% N41:130 % 0 30 5 30 2291 11737 100 -16 -68 0
% N41:140 % -28880 9190 14028 2291 16383 0 0 13000 11000 10000
% N41:150 % 8000 7000 6500 0 0 0 0 0 6500 6500
% N41:160 % 0 14000 14000 1370 224 1000 1000 150 0 100
% N41:170 % 120 0 40 15 0 0 0 0 0 0
DATA N42
% N42:0 % -32239 21248 14028 152 250 0 0 16383 0 0
% N42:10 % 0 30 5 30 2291 11737 100 -16 -68 0
% N42:20 % -28880 9190 14028 0 16383 0 0 35 35 35
% N42:30 % 35 35 0 0 0 0 0 0 0 0
% N42:40 % 0 0 35 1370 0 1000 1000 150 0 110
% N42:50 % 100 0 25 25 0 0 0 0 0 0
% N42:60 % 529 21248 14028 152 250 0 0 16383 0 0
% N42:70 % 0 30 5 30 2291 11737 100 0 0 0
% N42:80 % 0 9190 14028 0 16383 0 0 35 35 35
% N42:90 % 35 35 0 0 0 0 0 0 0 0
% N42:100 % 0 0 35 1370 0 1000 1000 150 0 110
% N42:110 % 100 0 25 25 0 0 0 0 0 0
% N42:120 % -32239 21248 14028 152 250 0 0 16383 0 0
% N42:130 % 0 30 5 30 2291 11737 100 -16 -68 0
% N42:140 % -28880 9190 14028 2291 16383 0 0 10 10 10
% N42:150 % 10 10 0 0 0 0 0 0 0 0
% N42:160 % 0 0 10 1370 224 1000 1000 150 0 110
% N42:170 % 100 0 25 25 0 0 0 0 0 0
% N42:180 % -32239 21248 14028 152 250 0 0 16383 0 0
% N42:190 % 0 30 5 30 2291 11737 100 -16 -68 0
% N42:200 % -28880 9190 14028 0 16383 0 0 40 0 0
% N42:210 % 0 0 0 0 0 0 0 0 0 40
% N42:220 % 0 0 40 1370 0 1000 1000 150 0 110
% N42:230 % 100 0 25 25 0 0 0 0 0 0
DATA N43
% N43:0 % -32239 21248 14028 152 250 0 0 16383 0 0
% N43:10 % 0 30 5 30 2291 11737 100 -16 -68 0
% N43:20 % -28880 9190 14028 2291 16383 0 0 300 200 0
% N43:30 % 0 0 0 0 0 0 0 0 0 500
% N43:40 % 0 0 500 1370 224 1000 1000 150 0 65
% N43:50 % 60 0 100 100 0 0 0 0 0 500
% N43:60 % 21 0 8192 320 42 0 0 16383 0 0
% N43:70 % 0 30 5 30 0 0 0 0 0 0
% N43:80 % 0 0 0 7707 0 0 0 500 500 500
% N43:90 % 500 500 0 0 0 0 0 200 0 0
% N43:100 % 0 500 400 500 470 0 0 25 0 320
% N43:110 % 300 0 25 20 0 0 0 0 0 0
% N43:120 % 21 0 13106 80 107 0 0 16383 0 0
% N43:130 % 0 100 65 30 0 0 0 0 0 0
% N43:140 % 0 0 0 3916 0 0 0 800 800 900
% N43:150 % 700 700 0 0 0 0 0 0 0 800
% N43:160 % 0 900 0 800 239 0 0 64 0 80
% N43:170 % 60 0 64 100 0 0 0 0 0 0
% N43:180 % -32239 21248 14028 152 250 0 0 16383 0 0
% N43:190 % 0 30 5 30 2291 11737 100 -16 -68 0
% N43:200 % -28880 9190 14028 2291 16383 0 0 650 0 0
% N43:210 % 0 0 0 0 0 0 0 0 0 600
% N43:220 % 0 0 0 1370 224 1000 1000 150 0 65
% N43:230 % 60 0 100 100 0 0 0 0 0 0
DATA N44
% N44:0 % 21 0 2355 200 42 0 0 16383 0 0
% N44:10 % 0 30 5 30 0 0 0 0 0 0
% N44:20 % 0 0 0 3004 0 0 0 230 245 240
% N44:30 % 250 80 0 200 0 0 0 0 0 0
% N44:40 % 0 0 0 230 294 0 0 25 0 200
% N44:50 % 150 150 25 25 25 0 0 0 0 0
% N44:60 % -32239 21248 14028 152 250 0 0 16383 0 0
% N44:70 % 0 30 5 30 2291 11737 100 -16 -68 0
% N44:80 % -28880 9190 14028 0 16383 0 0 810 810 810
% N44:90 % 810 810 0 0 0 0 0 0 0 0
% N44:100 % 0 0 0 1370 0 1000 1000 150 0 110
% N44:110 % 140 0 15 15 0 0 0 0 0 0
% N44:120 % 1045 21248 14028 0 0 0 0 16383 0 0
% N44:130 % 0 30 5 30 0 0 0 0 0 0
% N44:140 % 0 2959 0 0 0 0 0 200 250 220
% N44:150 % 250 250 0 0 0 0 0 0 0 0
% N44:160 % 0 0 0 1370 0 0 0 0 0 200
% N44:170 % 150 150 25 25 25 0 0 0 0 0
% N44:180 % -32239 21248 14028 152 250 0 0 16383 0 0
% N44:190 % 0 30 5 30 2291 11737 100 -16 -68 0
% N44:200 % -28880 9190 14028 2291 16383 0 0 800 0 0
% N44:220 % 0 0 0 1370 224 1000 1000 150 0 100
% N44:230 % 120 0 40 15 0 0 0 0 0 0
DATA N45
% N45:20 % 0 0 0 0 0 0 0 250 0 0
% N45:30 % 0 0 0 0 0 0 0 0 0 850
% N45:40 % 0 0 850 0 0 0 0 0 0 110
% N45:50 % 140 0 15 15 0 0 0 0 0 0
% N45:60 % 17 0 7680 150 67 0 0 16383 0 0
% N45:70 % 0 100 0 30 0 0 0 0 0 0
% N45:80 % 0 0 0 2635 0 0 0 750 750 750
% N45:90 % 830 830 0 0 0 0 0 0 0 0
% N45:100 % 0 0 700 750 257 0 0 40 0 150
% N45:110 % 150 0 40 30 0 0 0 0 0 0
% N45:120 % 17 0 14233 300 25 0 0 16383 0 0
% N45:130 % 0 30 5 30 0 0 0 0 0 0
% N45:140 % 0 0 0 2468 0 0 0 1390 1040 1390
% N45:150 % 1370 950 0 20 0 0 0 0 1010 1380
% N45:160 % 1300 800 1050 1390 241 0 0 15 0 300
% N45:170 % 320 320 15 5 5 0 0 0 0 0
% N45:180 % -32239 21248 14028 152 250 0 0 16383 0 0
% N45:190 % 0 30 5 30 2291 11737 100 -16 -68 0
% N45:200 % -28880 9190 14028 2291 16383 0 0 950 950 950
% N45:210 % 950 950 0 0 0 0 0 0 0 200
% N45:220 % 0 0 0 1370 224 1000 1000 150 0 110
% N45:230 % 140 0 15 15 0 0 0 0 0 0
DATA N46
% N46:0 % -32239 21248 14028 152 250 0 0 16383 0 0
% N46:10 % 0 30 5 30 2291 11737 100 -16 -68 0
% N46:20 % -28880 9190 14028 2291 16383 0 0 0 0 0
% N46:40 % 0 0 0 1370 224 1000 1000 150 0 200
% N46:50 % 150 0 25 25 0 0 0 0 0 0
% N46:60 % -32239 21248 14028 152 250 0 0 16383 0 0
% N46:70 % 0 30 5 30 2291 11737 100 -16 -68 0
% N46:80 % -28880 9190 14028 2291 16383 0 0 10 20 10
% N46:90 % 10 10 0 0 0 0 800 0 0 114
% N46:100 % 0 0 114 1370 224 1000 1000 150 0 110
% N46:110 % 140 0 15 15 0 0 0 0 0 0
% N46:120 % -32239 21248 14028 152 250 0 0 16383 0 0
% N46:130 % 0 30 5 30 2291 11737 100 -16 -68 0
% N46:140 % -28880 9190 14028 0 16383 0 0 750 100 0
% N46:150 % 0 0 0 0 0 0 0 0 0 200
% N46:160 % 650 750 100 1370 0 1000 1000 150 0 110
% N46:170 % 140 0 15 15 0 0 0 0 0 0
% N46:180 % 21 0 8703 200 33 0 0 16383 0 0
% N46:190 % 0 30 5 30 0 0 0 0 0 0
% N46:200 % 0 0 0 2927 0 0 0 850 0 0
% N46:210 % 0 0 0 0 0 0 200 0 0 0
% N46:220 % 0 0 0 850 286 0 0 20 0 200
% N46:230 % 300 300 20 25 30 0 0 0 0 0
DATA N47
% N47:0 % 21 0 7680 200 25 0 0 16383 0 0
% N47:10 % 0 30 5 30 0 0 0 0 0 0
% N47:20 % 0 0 0 2938 0 0 0 750 0 0
% N47:30 % 0 0 0 0 0 0 550 0 0 750
% N47:40 % 0 0 0 750 287 0 0 15 0 200
% N47:50 % 250 270 15 15 15 0 0 0 0 0
% N47:60 % 1041 21248 14028 0 0 0 0 16383 0 0
% N47:70 % 0 30 5 30 16383 -16383 0 0 0 0
% N47:80 % 0 2955 0 0 0 0 0 750 750 750
% N47:90 % 750 750 0 0 0 0 0 0 0 0
% N47:100 % 0 0 0 1370 0 0 0 0 0 200
% N47:110 % 200 0 150 250 0 0 0 0 0 0
% N47:120 % 0 0 0 6548 0 0 0 0 0 0
% N47:140 % 0 0 0 0 0 0 0 0 0 639
% N47:180 % 1041 21248 14028 0 0 0 0 16383 0 0
% N47:190 % 0 30 5 30 2291 -2291 0 0 0 0
% N47:200 % 0 47 0 0 0 0 0 850 850 850
% N47:210 % 850 850 0 0 0 0 0 0 0 0
% N47:220 % 0 0 850 1370 0 0 0 0 0 150
% N47:230 % 150 0 150 150 0 0 0 0 0 0
DATA N48
% N48:40 % 0 0 0 0 0 0 0 0 0 500
% N48:50 % 500 0 30 30 0 0 0 0 0 0
% N48:80 % 0 0 0 0 0 0 0 1200 1200 1200
% N48:90 % 1200 1200 0 0 0 0 0 0 0 0
% N48:100 % 0 0 0 0 0 0 0 0 0 150
% N48:110 % 150 0 150 150 0 0 0 0 0 0
DATA B49
% B49:0 % 0X0000 0X0080 0X0088 0X0000 0X0000 0X0000 0X0000 0X0000 0X0000 0X0000
DATA N50
% N50:20 % 0 0 0 0 0 0 8 0 0 0
% N50:50 % 17 15 1 0 0 0 0 0 0 0
DATA N51
% N51:0 % -32768 0 0 0 0 0 0 8 0 0
% N51:10 % 0 20504 0 0 0 4 0 -990 12800 0
% N51:20 % 0 16426 0 0 0 0 0 1 0 1556
% N51:40 % 0 0 0 0 0 0 0 167 0 0
% N51:70 % 0 0 0 0 0 0 0 0 0 1
% N51:80 % 1 0 0 1 16 1 16 0 0 0
% N51:90 % 0 0 0 0 1 16 1 16 0 4
% N51:100 % 1 1 1 0 0 0 0 2 1 294
% N51:110 % 294 4 294 294 244 244 986 986 0 42
% N51:120 % 26 71 42 8 0 0 0 0 0 0
% N51:130 % 2 1 1 1 1 2 0 0 0 44
% N51:150 % 263 270 286 206 0 0 0 986 267 242
% N51:160 % 0 0 0 0 0 30 0 30 0 0
% N51:170 % 0 0 12689 12157 35 34 239 0 0 0
% N51:180 % 0 0 0 500 600 400 150 350 300 15
% N51:190 % 350 10 0 0 0 0 13 2 0 350
% N51:210 % 0 0 0 0 0 0 0 0 0 125
% N51:220 % 2 16 0 0 0 0 0 0 0 0
% N51:230 % 12 0 0 0 -90 0 0 0 0 -98
% N51:240 % 0 0 0 0 0 118 235 0 0 0
% N51:250 % -4 4 0 0 0 0
DATA N52
% N52:0 % 0 7 0 0 0 0 304 13 18 0
% N52:10 % 150 30001 0 0 0 0 0 0 0 0
% N52:30 % 10 0 15 0 0 0 0 0 0 0
% N52:40 % 0 1 0 0 0 0 0 0 0 0
% N52:60 % 2000 1 1 0 0 0 0 0 0 0
DATA B53
% B53:0 % 0X0002 0X0000 0X0000 0X0000 0X0000 0X0800 0X0000 0X0000 0X0000 0X4000
% B53:10 % 0X0001 0X0000 0X0000 0X0000 0X0000 0X0000 0X0800 0X4100 0X00A9 0X0000
% B53:20 % 0X0000 0X4000 0X8000 0X0000 0X0000 0X0000 0X0000 0X0000 0X0000 0X0000
DATA N54
% N54:0 % -24576 0 0 0 0 0 0 0 0 0
% N54:10 % 166 0 0 0 0 0 0 0 0 0
% N54:30 % 0 0 0 0 0 353 0 0 0 0
% N54:50 % -32768 0 0 0 0 0 0 0 0 0
DATA N60
% N60:0 % 8192 11 1 54 137 10 0 224 5 146
% N60:10 % 0 2 3072 0 0 0 0 0 0 0
% N60:20 % 0 12 1 54 137 10 0 0 5 0
% N60:40 % 8192 3 1 231 137 1 0 96 5 146
% N60:50 % 0 2 3072 0 0 0 0 0 0 0
% N60:60 % 0 14 1 54 137 10 0 0 5 0
% N60:100 % 8192 4 1 59 137 10 0 160 5 146
% N60:110 % 0 2 3072 0 0 0 0 0 0 0
% N60:140 % 8192 3 1 231 137 41 0 32 5 146
% N60:150 % 0 2 3072 0 0 0 0 0 0 0
% N60:200 % 8192 5 1 232 137 41 0 0 5 0
DATA N61
% N61:0 % 0 0 1 54 137 10 0 0 5 0
% N61:10 % 0 0 0 0 12337 12334 12334 12590 49 0
DATA N63
% N63:0 % 0 0 1 54 137 60 0 0 5 0
% N63:10 % 0 0 0 0 12337 12334 12334 12846 48 0
DATA N75
% N75:0 % 0 5 5 180 25 10 1800 200 0 0
% N75:10 % 60 400 450 0 0 0 0 0 0 0
% N75:20 % 0 600 0 3 287 20 0 0 0 83
% N75:40 % 0 277 95 285 0 0 0 0 0 0
% N75:50 % 0 0 320 1800 0 350 0 320 0 0
% N75:60 % 0 0 350 0 0 0 0 0 0 0
% N75:70 % 0 740 0 0 0 0 0 0 222 50
% N75:80 % 60 101 116 170 0 0 0 0 0 0
% N75:100 % 0 5 5 300 25 0 0 0 0 0
% N75:110 % 0 330 0 260 1800 0 0 0 0 0
% N75:120 % 0 330 30 0 235 1500 0 0 0 0
% N75:130 % 0 330 0 260 24 0 0 0 0 0
% N75:140 % 0 330 0 270 300 1800 330 600 0 0
% N75:150 % 0 10 12 16 20 0 0 0 0 0
DATA N76
% N76:0 % 0 0 0 5 15 30 15 30 0 0
% N76:10 % 5 15 30 15 30 0 0 0 0 0
DATA N77
% N77:0 % 0 100 5 15 3 40 15 3 0 0
% N77:10 % 0 50 0 0 0 0 0 0 0 0
% N77:20 % 0 0 0 0 0 5 100 40 0 0
% N77:30 % 0 0 0 0 0 4 100 40 0 0
% N77:40 % 0 0 0 0 0 4 100 40 0 0
% N77:50 % 0 0 0 0 0 4 100 40 0 0
% N77:60 % 0 0 0 0 0 5 100 40 0 0
DATA N78
% N78:0 % 0 101 102 103 104 112 113 114 147 0
% N78:40 % 0 0 0 0 0 0 0 0 0 147
DATA N79
% N79:0 % 0 10 11 12 13 20 60 120 70 0
DATA B84
% B84:0 % 0X0000 0X0000 0X0000 0X2000
DATA N89
% N89:0 % 0 1 11000 10000 8000 7000 6500 0 0 0
% N89:10 % 85 285 20 0 65 0 15 90 80 12
% N89:20 % 12 185 95 0 65 0 15 1 11 111
% N89:50 % 50 70 0 0 0 0 0 0 0 0
% N89:110 % 0 0 0 0 0 0 0 0 0 100
% N89:120 % 0 100 50 50 50 50 50 0 0 0
% N89:130 % 0 30 30 30 30 30 30 0 0 0
% N89:140 % 0 390 450 400 350 300 250 0 0 0
% N89:150 % 0 0 50 10 10 10 0 0 0 0
DATA N90
% N90:0 % 105 1500 1500 0 105 0 0 0 0 0
% N90:10 % 0 0 0 0 0 0 0 0 -877 -257
DATA N91
% N91:0 % 0 5 5 180 25 10 1800 200 0 0
% N91:10 % 60 400 450 0 0 0 0 0 0 0
% N91:20 % 0 600 0 3 287 20 0 0 0 83
% N91:40 % 0 277 95 285 0 0 0 0 0 0
% N91:50 % 0 0 320 1800 0 350 0 320 0 0
% N91:60 % 0 0 350 0 0 0 0 0 0 0
% N91:70 % 0 740 0 0 0 0 0 0 0 55
% N91:80 % 0 5 5 300 25 0 0 0 0 0
% N91:90 % 0 330 0 260 1800 0 0 0 0 0
% N91:100 % 0 330 30 0 235 1500 0 0 0 0
% N91:110 % 0 330 0 260 24 0 0 0 0 0
% N91:120 % 0 330 0 270 300 1800 330 600 0 0
% N91:130 % 0 10 12 16 20 0 0 0 0 0
% N91:140 % 0 13000 11000 10000 8000 7000 6500 0 0 0
% N91:150 % 0 13000 11000 10000 8000 7000 6500 0 0 0
% N91:160 % 0 0 0 5 15 30 15 30 0 0
% N91:170 % 5 15 30 15 30 0 0 0 0 0
% N91:180 % 0 100 5 15 3 40 15 3 0 0
% N91:190 % 20 25 25 30 0 0 0 0 500 400
% N91:200 % 100 100 100 100 150 70 0 620 0 0
% N91:210 % 4000 50 0 24000 400 0 100 0 7350 0
% N91:220 % 0 20000 20000 0 1600 0 100 0 0 0
% N91:230 % 10 50 50 50 50 30 30 0 0 0
% N91:240 % 0 300 300 300 300 300 300 0 500 500
DATA N92
% N92:0 % 750 400 370 280 600 500 930 770 500 550
% N92:10 % 500 0 10 10 10 10 0 0 770 750
% N92:30 % 1000 900 800 700 600 500 890 900 500 500
% N92:40 % 500 0 10 10 10 10 0 0 900 1000
% N92:60 % 935 712 630 420 500 500 950 950 530 510
% N92:70 % 500 0 10 10 10 10 0 0 950 935
% N92:80 % 0 15000 11000 10000 6600 7000 6500 8000 20000 0
% N92:90 % 1000 900 800 700 600 500 1000 1000 500 500
% N92:100 % 500 0 20 10 10 10 0 0 0 0
% N92:110 % 0 13000 11000 10000 8000 7000 6500 6500 14000 0
% N92:120 % 1000 900 800 700 600 500 700 1000 250 600
% N92:130 % 500 0 10 10 10 10 0 0 1000 480
% N92:150 % 950 900 800 700 600 500 760 820 500 200
% N92:160 % 500 0 10 10 10 10 0 0 820 680
% N92:200 % 1000 900 800 900 600 500 1000 1000 500 500
% N92:210 % 0 0 20 10 10 10 0 0 0 0
% N92:220 % 1000 900 800 900 600 500 1000 1000 500 500
% N92:230 % 0 0 20 10 10 10 0 0 0 0
% N92:240 % 0 2 4 0 0 0 0 0 0 0
DATA N93
% N93:0 % 750 600 700 700 700 700 950 950 530 460
% N93:10 % 0 0 20 10 10 10 0 0 0 0
% N93:20 % 660 430 700 700 700 700 750 750 450 450
% N93:30 % 0 0 20 10 10 10 0 0 0 0
% N93:40 % 700 700 700 700 700 700 700 700 700 700
% N93:50 % 0 0 20 10 10 10 0 0 0 0
% N93:60 % 1000 650 320 150 700 700 700 700 700 700
% N93:70 % 0 0 20 10 10 10 0 850 150 150
% N93:90 % 0 6000 6000 3600 1500 0 0 0 0 0
% N93:100 % 0 285 384 424 623 900 950 0 0 0
% N93:110 % 0 20 30 38 51 40 45 0 0 0
% N93:120 % 0 65 86 89 100 50 60 0 0 0
% N93:140 % 0 15 20 23 34 100 120 0 0 0
% N93:150 % 0 285 389 428 648 900 950 0 0 0
% N93:160 % 0 185 250 356 410 800 900 0 0 0
% N93:170 % 0 95 125 178 253 30 35 0 0 0
% N93:180 % 0 65 86 89 100 50 60 0 0 0
% N93:190 % 0 0 0 0 0 25 0 0 0 0
% N93:200 % 0 15 20 23 34 100 120 0 0 0
% N93:210 % 320 320 0 0 0 0 320 320 0 0
% N93:220 % 330 330 330 330 600 500 400 400 400 500
% N93:230 % 4 160 3 120 3 120 3 120 4 160
% N93:240 % 0 12 20 24 41 900 12 20 24 41
DATA N94
% N94:0 % 50 50 1 1 0 0 0 0 0 0
% N94:10 % 50 50 1 1 0 0 0 0 0 0
% N94:20 % 50 50 1 1 0 10 20 10 20 0
% N94:30 % 50 50 1 1 0 10 20 10 20 0
% N94:40 % 50 50 1 1 0 0 0 0 0 0
% N94:50 % 50 50 1 1 0 0 0 0 0 0
% N94:60 % 50 50 1 1 0 0 0 0 0 0
% N94:70 % 0 0 0 0 5 1 600 100 100 0
% N94:80 % 50 50 1 1 5 1 1200 100 100 0
% N94:90 % 0 0 0 0 5 1 900 0 0 0
% N94:100 % 0 0 0 0 5 1 0 0 0 0
% N94:110 % 0 0 0 0 0 0 950 0 0 0
% N94:120 % 0 30 41 45 68 73 80 0 0 0
% N94:130 % 0 350 1250 950 950 850 900 0 0 0
% N94:140 % 0 1000 0 0 0 0 0 0 0 0
% N94:150 % 0 500 0 0 0 0 0 0 0 0
% N94:160 % 0 900 0 0 0 0 0 0 0 0
% N94:170 % 0 400 0 0 0 0 0 0 0 0
% N94:180 % 0 30 41 45 68 70 80 0 0 0
% N94:200 % 1000 900 800 700 600 500 1000 1000 500 500
% N94:210 % 0 0 20 10 10 10 0 0 0 0
% N94:220 % 8657 13041 2510 0 0 0 0 0 0 0
% N94:230 % 22936 30001 3998 0 0 0 0 23 55 0
% N94:240 % 0 50 101 116 185 0 0 0 0 0
DATA N95
% N95:0 % 200 100 60 0 0 0 0 0 0 0
% N95:10 % 0 480 600 550 1000 1000 0 0 0 0
% N95:20 % 0 300 300 300 900 900 0 0 0 0
% N95:30 % 0 200 200 200 800 800 0 0 0 0
% N95:40 % 0 40 50 100 700 700 0 0 0 0
% N95:50 % 0 600 600 600 600 600 0 0 0 0
% N95:60 % 0 500 500 500 500 500 0 0 0 0
% N95:70 % 500 600 500 250 450 0 0 0 0 0
% N95:80 % 0 700 100 650 10 10 0 0 0 0
% N95:90 % 350 350 350 300 300 0 0 0 0 0
% N95:100 % 0 0 100 10 10 10 0 0 0 0
% N95:110 % 0 680 510 510 1000 1000 0 0 0 0
% N95:120 % 0 400 400 400 900 900 0 0 0 0
% N95:130 % 0 250 250 250 800 800 0 0 0 0
% N95:140 % 0 380 0 0 700 700 0 0 0 0
% N95:150 % 0 600 600 600 600 600 0 0 0 0
% N95:160 % 0 500 500 500 500 500 0 0 0 0
% N95:170 % 0 90 125 178 205 0 0 0 0 85
% N95:180 % 0 80 95 100 157 0 0 0 0 0
DATA N105
% N105:0 % 2 2 -32767 -32767 -32767 2 -32767 4098 2 2
% N105:10 % 2 -32767 0 0 0 0 0 0 0 0
